TYPE M2Tabs :
(
	OVERVIEW := 0,
    AXES := 1,
    TECHNICAL := 2,
    IO := 3,
    CONFIG := 4
);
END_TYPE

(* stored: Version 1.1.0.1, ProductVersion 3.1.4018.5
   DUT M2Tabs: Id {0ee6456e-6f84-44da-8594-994394862708} *)
